PROGRAM Monitoring
VAR	

END_VAR

VAR RETAIN PERSISTENT
	ShapeMonitor01					:	ShapeMonitor;
END_VAR

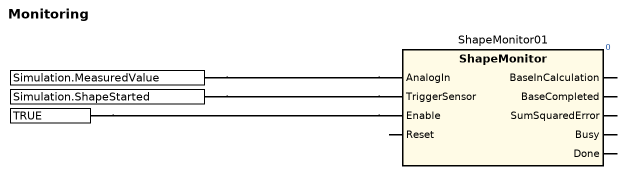
ShapeMonitor01(
    AnalogIn := Simulation.MeasuredValue,
    TriggerSensor := Simulation.ShapeStarted,
    Enable := TRUE); // ShapeMonitor

END_PROGRAM

(* stored: Version 1.1.0.1, ProductVersion 3.1.4024.12
   POU Monitoring: Id {57c128e3-2ec7-49c2-a729-7462493cc98a}, SpecialFunc None *)
